FUNCTION_BLOCK Skill_R_P2P EXTENDS FB_SkillBasis
VAR_INPUT
	// Objekt
	Roboter				:I_Objekt_Roboter;
	
	// Prozessparameter
	Position			:sPositionValues;
	Geschw				:LREAL;
	Beschl				:LREAL;
	PosTyp				:eRobPosType;
	MoveTyp				:eRobMoveType;	
END_VAR
VAR_OUTPUT
END_VAR
VAR
	Prozessparameter	:sRoboterProzessVariablen; 
END_VAR

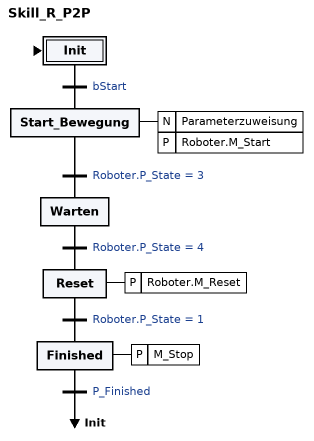
INITIAL_STEP Init:
END_STEP
TRANSITION FROM Init TO Start_Bewegung
    := bStart;
END_TRANSITION
STEP Start_Bewegung:
    Parameterzuweisung(N);
    Roboter.M_Start(P);
END_STEP
TRANSITION FROM Start_Bewegung TO Warten
    := Roboter.P_State = 3;
END_TRANSITION
STEP Warten:
END_STEP
TRANSITION FROM Warten TO Reset
    := Roboter.P_State = 4;
END_TRANSITION
STEP Reset:
    Roboter.M_Reset(P);
END_STEP
TRANSITION FROM Reset TO Finished
    := Roboter.P_State = 1;
END_TRANSITION
STEP Finished:
    M_Stop(P);
END_STEP
TRANSITION FROM Finished TO Init
    := P_Finished;
END_TRANSITION

ACTION Parameterzuweisung:
// Variablenzuweisung
Prozessparameter.q1 := Position.q1;
Prozessparameter.q2 := Position.q2;
Prozessparameter.q3 := Position.q3;
Prozessparameter.q4 := Position.q4;
Prozessparameter.q5 := Position.q5;
Prozessparameter.q6 := Position.q6;
Prozessparameter.v := Geschw;
Prozessparameter.a := Beschl;
Prozessparameter.MoveTyp := MoveTyp;
Prozessparameter.PosTyp := PosTyp;

//Zuweisung an Objekt
Roboter.P_Prozessparameter := Prozessparameter;
END_ACTION

END_FUNCTION_BLOCK

(* stored: Version 1.1.0.1
   POU Skill_R_P2P: Id {c4b5a27c-d27f-4f86-9fb5-58e997a56248}, SpecialFunc None
   Action Parameterzuweisung: Id {25868ac2-53a0-4200-9692-b60c31dcfa2f} *)
